% RSLogix 500 project P2_KOBIERSKI_M_v1.RSS, saved by version 8.30.00.16 %
PROJECT "UNTITLED"    % processor: Bul.1763 MicroLogix 1100 Series B %

PROGRAM FILES
  LAD 2 "MAIN"  3 rungs
  LAD 3 "IO"  8 rungs
  LAD 4 "CTRL"  6 rungs

DATA FILES
  O0 OUTPUT  4 elements
  I1 INPUT  6 elements
  S2 STATUS  66 elements
  B3 BINARY  3 elements
  T4 TIMER  2 elements
  C5 COUNTER  1 elements
  R6 CONTROL  1 elements
  N7 INTEGER  1 elements
  F8 FLOAT  1 elements

LADDER 2 "MAIN"
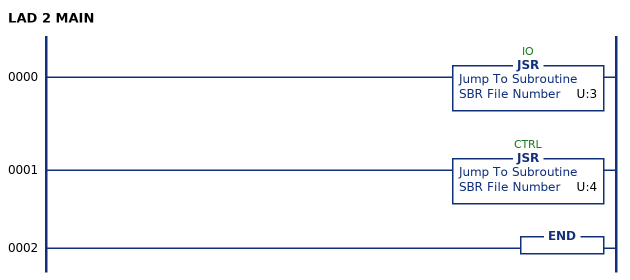
% Rung: 0 %
SOR JSR U:3 EOR
%   U:3  "IO" %
% Rung: 1 %
SOR JSR U:4 EOR
%   U:4  "CTRL" %
% Rung: 2 %
SOR END EOR

LADDER 3 "IO"
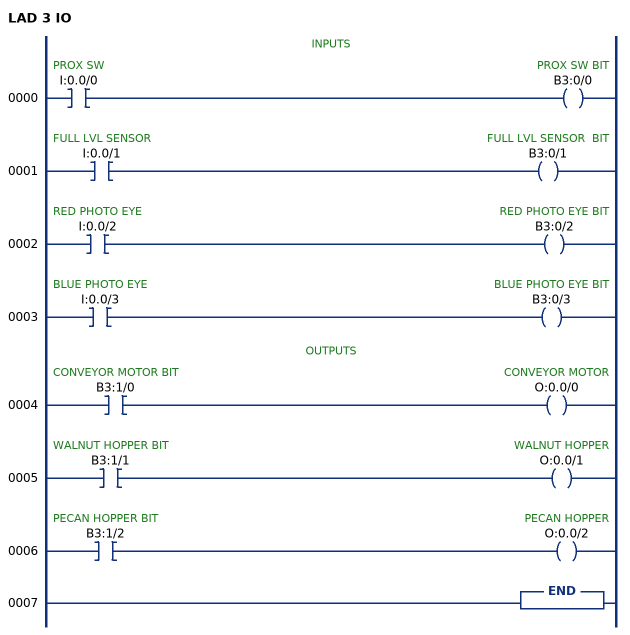
% Rung: 0 %
% INPUTS %
SOR XIC I:0.0/0 OTE B3:0/0 EOR
%   I:0.0/0  "PROX SW" %
%   B3:0/0  "PROX SW BIT" %
% Rung: 1 %
SOR XIC I:0.0/1 OTE B3:0/1 EOR
%   I:0.0/1  "FULL LVL SENSOR" %
%   B3:0/1  "FULL LVL SENSOR  BIT" %
% Rung: 2 %
SOR XIC I:0.0/2 OTE B3:0/2 EOR
%   I:0.0/2  "RED PHOTO EYE" %
%   B3:0/2  "RED PHOTO EYE BIT" %
% Rung: 3 %
SOR XIC I:0.0/3 OTE B3:0/3 EOR
%   I:0.0/3  "BLUE PHOTO EYE" %
%   B3:0/3  "BLUE PHOTO EYE BIT" %
% Rung: 4 %
% OUTPUTS %
SOR XIC B3:1/0 OTE O:0.0/0 EOR
%   B3:1/0  "CONVEYOR MOTOR BIT" %
%   O:0.0/0  "CONVEYOR MOTOR" %
% Rung: 5 %
SOR XIC B3:1/1 OTE O:0.0/1 EOR
%   B3:1/1  "WALNUT HOPPER BIT" %
%   O:0.0/1  "WALNUT HOPPER" %
% Rung: 6 %
SOR XIC B3:1/2 OTE O:0.0/2 EOR
%   B3:1/2  "PECAN HOPPER BIT" %
%   O:0.0/2  "PECAN HOPPER" %
% Rung: 7 %
SOR END EOR

LADDER 4 "CTRL"
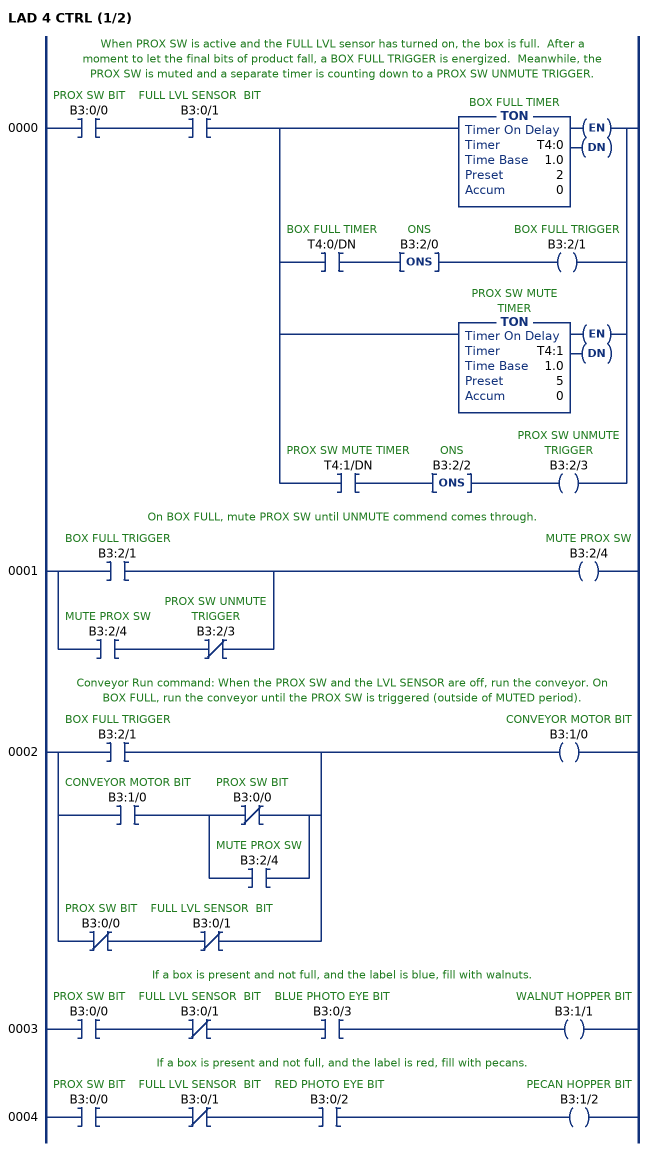
% Rung: 0 %
% When PROX SW is active and the FULL LVL sensor has turned on, the box is full.  After a moment to let the final bits of product fall, a BOX FULL TRIGGER is energized.  Meanwhile, the PROX SW is muted and a separate timer is counting down to a PROX SW UNMUTE TRIGGER. %
SOR XIC B3:0/0 XIC B3:0/1 BST TON T4:0 1.0 2 0 NXB XIC T4:0/DN ONS B3:2/0 OTE B3:2/1 NXB TON T4:1 1.0 5 0 NXB XIC T4:1/DN ONS B3:2/2 OTE B3:2/3 BND EOR
%   B3:0/0  "PROX SW BIT" %
%   B3:0/1  "FULL LVL SENSOR  BIT" %
%   T4:0  "BOX FULL TIMER" %
%   B3:2/0  "ONS" %
%   B3:2/1  "BOX FULL TRIGGER" %
%   T4:1  "PROX SW MUTE TIMER" %
%   B3:2/2  "ONS" %
%   B3:2/3  "PROX SW UNMUTE TRIGGER" %
% Rung: 1 %
% On BOX FULL, mute PROX SW until UNMUTE commend comes through. %
SOR BST XIC B3:2/1 NXB XIC B3:2/4 XIO B3:2/3 BND OTE B3:2/4 EOR
%   B3:2/1  "BOX FULL TRIGGER" %
%   B3:2/4  "MUTE PROX SW" %
%   B3:2/3  "PROX SW UNMUTE TRIGGER" %
% Rung: 2 %
% Conveyor Run command: When the PROX SW and the LVL SENSOR are off, run the conveyor. On BOX FULL, run the conveyor until the PROX SW is triggered (outside of MUTED period). %
SOR BST XIC B3:2/1 NXB BST XIC B3:1/0 BST XIO B3:0/0 NXB XIC B3:2/4 BND NXB XIO B3:0/0 XIO B3:0/1 BND BND OTE B3:1/0 EOR
%   B3:2/1  "BOX FULL TRIGGER" %
%   B3:1/0  "CONVEYOR MOTOR BIT" %
%   B3:0/0  "PROX SW BIT" %
%   B3:2/4  "MUTE PROX SW" %
%   B3:0/1  "FULL LVL SENSOR  BIT" %
% Rung: 3 %
% If a box is present and not full, and the label is blue, fill with walnuts. %
SOR XIC B3:0/0 XIO B3:0/1 XIC B3:0/3 OTE B3:1/1 EOR
%   B3:0/0  "PROX SW BIT" %
%   B3:0/1  "FULL LVL SENSOR  BIT" %
%   B3:0/3  "BLUE PHOTO EYE BIT" %
%   B3:1/1  "WALNUT HOPPER BIT" %
% Rung: 4 %
% If a box is present and not full, and the label is red, fill with pecans. %
SOR XIC B3:0/0 XIO B3:0/1 XIC B3:0/2 OTE B3:1/2 EOR
%   B3:0/0  "PROX SW BIT" %
%   B3:0/1  "FULL LVL SENSOR  BIT" %
%   B3:0/2  "RED PHOTO EYE BIT" %
%   B3:1/2  "PECAN HOPPER BIT" %

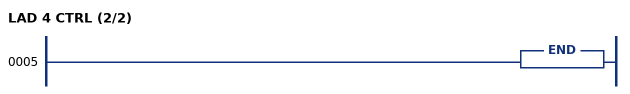
% Rung: 5 %
SOR END EOR

COMMENTS NOT ATTACHED TO A CURRENT RUNG
  B3:2/1: Once a box is full, delay a moment to catch and final falling product then trigger the BOX FULL signal.
  T4:1: When PROX SW and FULL LVL SENSOR are both on, 1) short delay to catch final falling product; 2) longer delay muting the PROX SW bit to let the box pass.

DATA TABLE (non-zero values as saved)
DATA T4
% .PRE .ACC %
% T4:0 % 2 0
% T4:1 % 5 0
